# EPICS substitutions: example_ioc/lexiumApp/Db/clearlock.substitutions
file "db/clearlock.db"
{
pattern
{Sys,                   Dev,        PORT  }
{"XF:12ID1-ES", "{Slt1-Ax:T}",   P1  }
{"XF:12ID1-ES", "{Slt1-Ax:B}",   P2  }
{"XF:12ID1-ES", "{Slt1-Ax:I}",   P3  }
{"XF:12ID1-ES", "{Slt1-Ax:O}",   P4  }
}
